FUNCTION_BLOCK FB_StateStill
VAR_IN_OUT
	stAxis  	: ARRAY [GVL.cXP .. GVL.cXM] OF ST_AxisGroup;
	bTopEntry	: BOOL;
END_VAR
VAR_INPUT
	eCommand			: E_Commands;
	stChangeAxisEnable	: ST_ChangeAxisEnable;
	stChangeBrakeState	: ST_ChangeBrakeState;
	stClearAllFaults	: ST_ClearAllFaults;
	stClearAxisFaults	: ST_ClearAxisFaults;
	stDisableAllAxes	: ST_DisableAllAxes;
	stEnableAllAxes		: ST_EnableAllAxes;
END_VAR
VAR_OUTPUT
	bBusy	: BOOL;
END_VAR
VAR
	//state-machine
	nCurrentState	: INT;
	nNextState		: INT;
END_VAR


IF bTopEntry = TRUE THEN
	bTopEntry := FALSE;
	bBusy := TRUE;
END_IF	

IF eCommand = E_Commands.clearAllFaults THEN
	nNextState := 1000;
ELSIF eCommand = E_Commands.changeAxisEnable THEN
	nNextState := 1010	;
ELSIF eCommand = E_Commands.clearAxisFaults THEN
	nNextState := 1020;
ELSIF eCommand = E_Commands.enableAllAxes THEN
	nNextState := 1030;
ELSIF eCommand = E_Commands.disableAllAxes THEN
	nNextState := 1040;
ELSIF eCommand = E_Commands.changeBrakeState THEN
	nNextState := 1050;
END_IF

nCurrentState := nNextState;

CASE nCurrentState OF

	1000:
		stAxis[GVL.cXM].mcReset(Axis:=stAxis[GVL.cXM].axisRef, Execute:=TRUE);
		stAxis[GVL.cXM].mcReset(Axis:=stAxis[GVL.cXM].axisRef, Execute:=TRUE);
		IF stAxis[GVL.cXP].mcReset.Done AND stAxis[GVL.cXM].mcReset.Done THEN
			stAxis[GVL.cXM].mcReset(Axis:=stAxis[GVL.cXM].axisRef, Execute:=FALSE);
			stAxis[GVL.cXM].mcReset(Axis:=stAxis[GVL.cXM].axisRef, Execute:=FALSE);
			nNextState := 2000; 
		END_IF
		
	1010:	
		stAxis[stChangeAxisEnable.axisIndex].mcPower(Axis:=stAxis[stChangeAxisEnable.axisIndex].axisRef,
			 Enable:=stChangeAxisEnable.enabled, Enable_Positive:=stChangeAxisEnable.enabled, Enable_Negative:=stChangeAxisEnable.enabled);
		//nNextState := 2000; 

	1020:	
		stAxis[stClearAxisFaults.axisIndex].mcReset(Axis:=stAxis[stClearAxisFaults.axisIndex].axisRef, Execute:=TRUE);
		IF stAxis[stClearAxisFaults.axisIndex].mcReset.Done THEN
			stAxis[stClearAxisFaults.axisIndex].mcReset(Axis:=stAxis[stClearAxisFaults.axisIndex].axisRef, Execute:=FALSE);
			nNextState := 2000; 
		END_IF

	1030:
		stAxis[GVL.cXP].mcPower(Axis:=stAxis[GVL.cXP].axisRef, Enable:=TRUE, Enable_Positive:=TRUE, Enable_Negative:=TRUE);
		stAxis[GVL.cXM].mcPower(Axis:=stAxis[GVL.cXM].axisRef, Enable:=TRUE, Enable_Positive:=TRUE, Enable_Negative:=TRUE);
		nNextState := 2000; 

	1040:	
		stAxis[GVL.cXP].mcPower(Axis:=stAxis[GVL.cXP].axisRef, Enable:=FALSE, Enable_Positive:=FALSE, Enable_Negative:=FALSE);
		stAxis[GVL.cXM].mcPower(Axis:=stAxis[GVL.cXM].axisRef, Enable:=FALSE, Enable_Positive:=FALSE, Enable_Negative:=FALSE);
		nNextState := 2000; 
		
	1050:
		stAxis[stChangeBrakeState.axisIndex].bBrake := NOT stChangeBrakeState.state;
		nNextState := 2000; 

	2000:
		bBusy := FALSE;
	
END_CASE

END_FUNCTION_BLOCK

(* stored: Version 1.1.0.1, ProductVersion 3.1.4020.12
   POU FB_StateStill: Id {fac21632-7010-4c07-91b9-f12f78686b07}, SpecialFunc None *)
